// TIA Portal project "les1" (V14)

(* hardware
DEVICE "S7-1200 station_1"  S7-1200 Station
   slot 0: "Rack_0"  S7-1200 Rack  Rack  V1.0
   slot 1: "PLC_1"  CPU 1214C DC/DC/DC  6ES7 214-1AG40-0XB0  V4.2
*)

// ===== PLC "PLC_1"  CPU 1214C DC/DC/DC =====

VAR_GLOBAL   // PLC tag table "Default tag table"
   "beginsensor" AT %I0.0 : Bool;
   "sensor" AT %I0.1 : Bool;
   "out1" AT %Q0.2 : Bool;
   "noodknop" AT %I0.3 : Bool;
   "stop" AT %I0.4 : Bool;
   "tag5" AT %I0.5 : Bool;
   "tag6" AT %I0.6 : Bool;
   "tag" AT %I0.7 : Bool;
   "tag8" AT %I1.0 : Bool;
   "tag9" AT %I1.1 : Bool;
   "tag10" AT %I1.2 : Bool;
   "tag11" AT %I1.3 : Bool;
   "tag12" AT %I1.4 : Bool;
   "tag13" AT %I1.5 : Bool;
END_VAR

// folder: System blocks/Program resources

DATA_BLOCK "IEC_Counter_0_DB"   // DB1
{ S7_Optimized_Access := 'TRUE' }
AUTHOR : Simatic
FAMILY : IEC
NAME : CNTR
VERSION : 1.0
// stored: InstanceOfName IEC_COUNTER
"IEC_COUNTER"
BEGIN
END_DATA_BLOCK

// folder: (top level)

ORGANIZATION_BLOCK "Main"   // OB1, LAD, ProgramCycle
TITLE = "Main Program Sweep (Cycle)"
{ S7_Optimized_Access := 'TRUE' }
VERSION : 0.1
   VAR_INPUT
      Initial_Call : Bool;   // Initial call of this OB
      Remanence : Bool;   // =True, if remanent data are available
   END_VAR
   VAR_TEMP   // added for the SCL form of the ladder/FBD networks
      _w1 : Bool;
   END_VAR
BEGIN

REGION Network 1
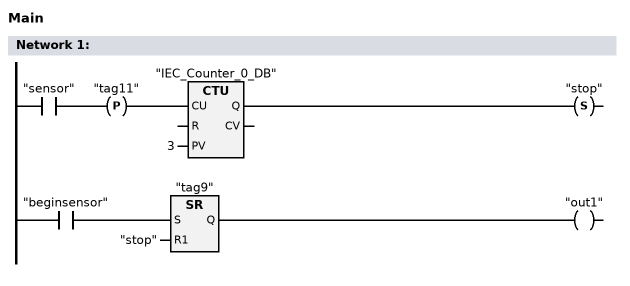
   #_w1 := "sensor" AND NOT "tag11";   // rising edge
   "tag11" := "sensor";
   "IEC_Counter_0_DB".CTU(CU := #_w1, PV := 3);
   IF "IEC_Counter_0_DB".Q THEN "stop" := TRUE; END_IF;
   IF "beginsensor" THEN
       "tag9" := TRUE;   // SR flip-flop
   END_IF;
   IF "stop" THEN "tag9" := FALSE; END_IF;
   "out1" := "tag9";
END_REGION
END_ORGANIZATION_BLOCK